{attribute 'qualified_only'}
//{attribute 'strict'}
{attribute 'to_string'}
TYPE eStationNo_1 :
(
	Station1 := 1,
	Station2 := 2,
	Station3 := 3,
	Station4 := 4,
	Station5 := 5,
	Station6 := 6,
	Station7 := 7
)DINT;
END_TYPE

(* stored: Version 1.1.0.1, ProductVersion 3.1.4024.3
   DUT eStationNo_1: Id {d42affa0-8506-463a-a501-a320e2ec7cbb} *)
